// TIA Portal V15.1 export
// export: Created 2024-05-17T05:38:43.2423617Z, ExportSetting WithDefaults, DisplayName Totally Integrated Automation Portal, DisplayVersion V15.1 Update 5, DisplayName TIA Portal Openness, DisplayVersion V15.1 Update 5, DisplayName SINAMICS Startdrive Advanced, DisplayVersion V15.1, DisplayName G130, G150, S120, S150, SINAMICS MV, S210, DisplayVersion V15.1, DisplayName G110M, G120, G120C, G120D, G120P, DisplayVersion V15.1, DisplayName STEP 7 Professional, DisplayVersion V15.1 Update 5, DisplayName STEP 7 Safety, DisplayVersion V15.1, DisplayName WinCC Professional, DisplayVersion V15.1 Update 5, DisplayName SIMATIC Visualization Architect, DisplayVersion V15.1
FUNCTION "LGBShuttle5Pos2S-MoviFitFCPN-Config" : Void   // FC6696, FBD
TITLE = LMoveEPos-Config / LGBShuttle5Pos2S-MoviFitFCPN-Config
{ S7_Optimized_Access := 'FALSE' }
AUTHOR : VCC
FAMILY : Config
VERSION : 0.0.0.0
// =============================================================================
// Configuration MoveUnitEpos
// =============================================================================
// ============================================================================
// Configuration MoveUnitEpos
// ============================================================================
// stored: AutoNumber false, IsIECCheckEnabled false, SetENOAutomatically False, UDAEnableTagReadback false
   VAR_INPUT
      C_ForceManual : Bool;   // Force Manual Enabled
      C_AlarmResetUsed : Bool;   // Set position / If true, the Alarms will be stored untill reseted
      C_EnableMemBegin : Bool;   // Reset position / Enable memory Begin (Command Request is memorised until pos reached)
      C_EnIntlkAlm : Bool;   // Active / Enable interlock Alarm
      C_KeepPosition : Bool;   // Invisible / If true, the last position shall be kept ON and checked
      C_EnAlmOvertime : Bool;   // Object out of use / Enable Alarm
      C_InitDirection : Bool;   // Initial direction
      C_EnablePos1 : Bool;   // Position 1 used / Pos 1 used
      C_EnablePos2 : Bool;   // Position 2 used / Pos 2 used
      C_EnablePos3 : Bool;   // Position 3 used / Pos 3 used
      C_EnablePos4 : Bool;   // Position 4 used / Pos 4 used
      C_EnablePos5 : Bool;   // Position 5 used / Pos 4 used
      C_EnablePosMaint : Bool;   // Position Maintenance used / Pos 4 used
      C_SetHigherEncValue : Bool;   // Set direction to get HIGHER Encoder value
      C_OverTravelSetUsed : Bool;   // Overtravel set used
      C_OverTravelResUsed : Bool;   // Overtravel reset used
      C_MotorProtectionNc : Bool;   // Motor Protection NC contact
      C_MotorProtectionUsed : Bool;   // Motor Protection used
      C_MotionStopUsed : Bool;   // Motion Stop used
      C_HartingPlug400VNc : Bool;   // Motor Protection NC contact / Harting plug 400V NC contact
      C_HartingPlug400VUsed : Bool;   // Motor Protection used / Harting plug 400V used
      C_HartingPlug24VNc : Bool;   // Motor Protection NC contact / Harting plug 24V NC contact
      C_HartingPlug24VUsed : Bool;   // Motor Protection used / Harting plug 24V used
      C_EnableAlarmHW : Bool;   // Enable Alarm hardware (e.g. safetyswitch, motorprotector, detections)
      C_ReleaseBrakeUsed : Bool;   // Release brake used
      C_WhichPosIsHomePos : DInt;   // Which position is home position
      C_Pos1 : DInt;   // Position Stop 1
      C_Pos2 : DInt;   // Position Stop 2
      C_Pos3 : DInt;   // Position Stop 3
      C_Pos4 : DInt;   // Position Stop 4
      C_Pos5 : DInt;   // Position Stop 5 / Position Stop 4
      C_PosMaint : DInt;   // Maintenance Position
      C_Diff_HH_LL : DInt;   // Difference HH / LL
      C_Diff_H_L : DInt;   // Difference H / L
      C_RunTimeMaxSetWarn : DInt;   // Maximum Time (x1ms) that the function may run (create Overtime)
      C_RunTimeMaxSetAlarm : DInt;   // Maximum Time (x1ms) that the function may run (create Overtime)
      C_RunTimeMaxResWarn : DInt;   // Maximum Time (x1ms) that the function may run (create Overtime)
      C_RunTimeMaxResAlarm : DInt;   // Maximum Time (x1ms) that the function may run (create Overtime)
      C_TimeAlmFilt : DInt;   // Timer before any actuator Alarm will be active (welding..)
      C_Ramp : Time;   // Reference value for speed, stored in P2000 ot the SINAMICS / Configuration
      C_ReferenceDriveCurrent : Real;   // Drive reference current / Reference current of the drive
      C_ReferenceMotorCurrent : Real;   // Motor reference current / Reference current of the motor
      C_ReferenceMotorRPM : Real;   // Reference RPM of the motor
      C_RatioGearbox : Real;   // Acceleration in m/s²
      C_Diameter : Real;   // Diameter in mm
      C_Acceleration : Real;   // Ratio Gearbox <-> Motor
      C_HWSubInput : HW_SUBMODULE;   // I/O
      C_HWSubOutput : HW_SUBMODULE;   // I/O
      C_HWSubInputStatus : HW_SUBMODULE;   // I/O
   END_VAR
   VAR_IN_OUT
      IO_Config : "Shuttle5Pos2S-MoviFitFCPNConfig";   // Config
   END_VAR
BEGIN

REGION Network 1: **** 1 - Inputs **** Configuration / **** 1 - Inputs **** Move Bit Config
   // Configuration
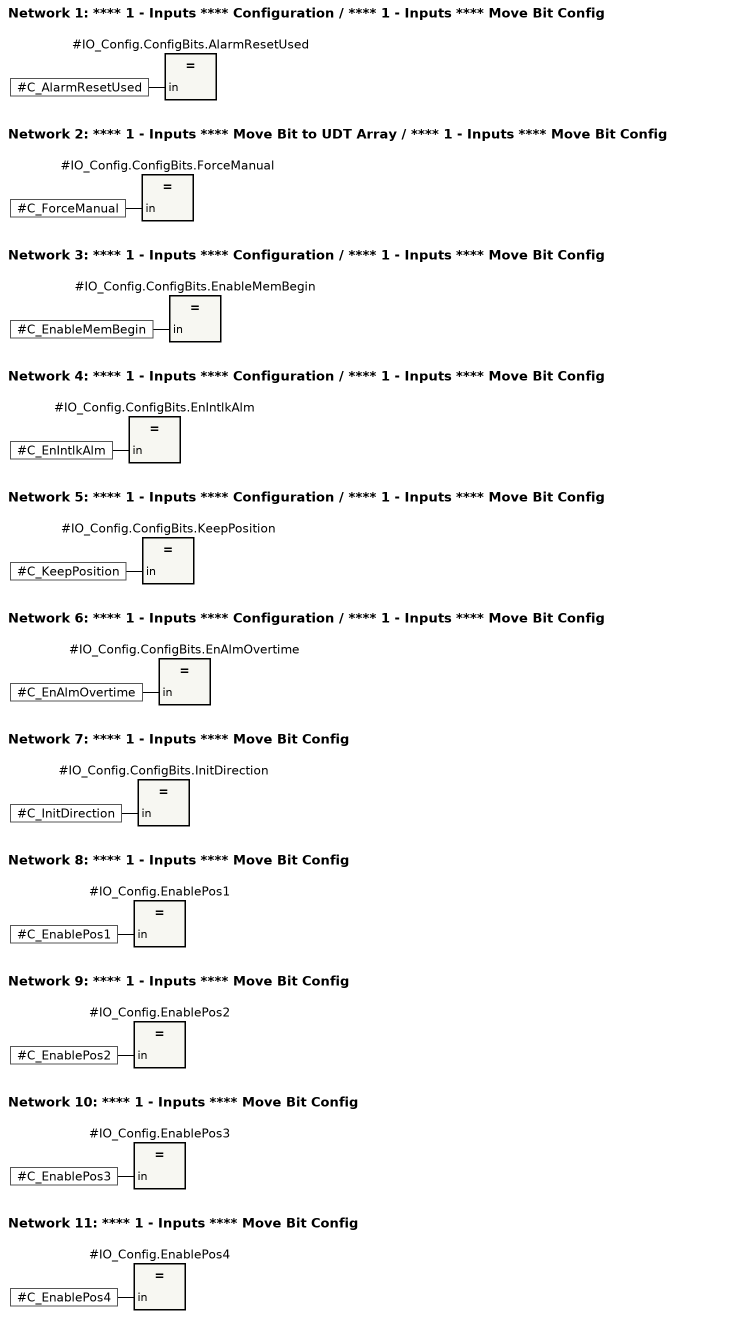
   #IO_Config.ConfigBits.AlarmResetUsed := #C_AlarmResetUsed;
END_REGION

REGION Network 2: **** 1 - Inputs **** Move Bit to UDT Array / **** 1 - Inputs **** Move Bit Config
   // Move Bit  to UDT Array
   #IO_Config.ConfigBits.ForceManual := #C_ForceManual;
END_REGION

REGION Network 3: **** 1 - Inputs **** Configuration / **** 1 - Inputs **** Move Bit Config
   // Configuration
   #IO_Config.ConfigBits.EnableMemBegin := #C_EnableMemBegin;
END_REGION

REGION Network 4: **** 1 - Inputs **** Configuration / **** 1 - Inputs **** Move Bit Config
   // Configuration
   #IO_Config.ConfigBits.EnIntlkAlm := #C_EnIntlkAlm;
END_REGION

REGION Network 5: **** 1 - Inputs **** Configuration / **** 1 - Inputs **** Move Bit Config
   // Configuration
   #IO_Config.ConfigBits.KeepPosition := #C_KeepPosition;
END_REGION

REGION Network 6: **** 1 - Inputs **** Configuration / **** 1 - Inputs **** Move Bit Config
   // Configuration
   #IO_Config.ConfigBits.EnAlmOvertime := #C_EnAlmOvertime;
END_REGION

REGION Network 7: **** 1 - Inputs **** Move Bit Config
   // Move Bit Config
   #IO_Config.ConfigBits.InitDirection := #C_InitDirection;
END_REGION

REGION Network 8: **** 1 - Inputs **** Move Bit Config
   // Move Bit Config
   #IO_Config.EnablePos1 := #C_EnablePos1;
END_REGION

REGION Network 9: **** 1 - Inputs **** Move Bit Config
   // Move Bit Config
   #IO_Config.EnablePos2 := #C_EnablePos2;
END_REGION

REGION Network 10: **** 1 - Inputs **** Move Bit Config
   // Move Bit Config
   #IO_Config.EnablePos3 := #C_EnablePos3;
END_REGION

REGION Network 11: **** 1 - Inputs **** Move Bit Config
   // Move Bit Config
   #IO_Config.EnablePos4 := #C_EnablePos4;
END_REGION

REGION Network 12: **** 1 - Inputs **** Move Bit Config
   // Move Bit Config
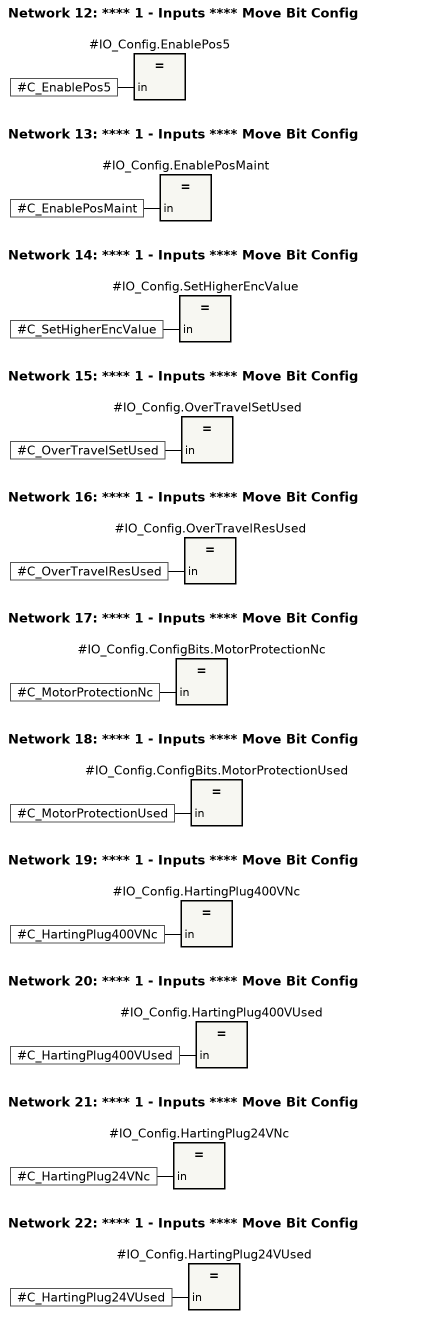
   #IO_Config.EnablePos5 := #C_EnablePos5;
END_REGION

REGION Network 13: **** 1 - Inputs **** Move Bit Config
   // Move Bit Config
   #IO_Config.EnablePosMaint := #C_EnablePosMaint;
END_REGION

REGION Network 14: **** 1 - Inputs **** Move Bit Config
   // Move Bit Config
   #IO_Config.SetHigherEncValue := #C_SetHigherEncValue;
END_REGION

REGION Network 15: **** 1 - Inputs **** Move Bit Config
   #IO_Config.OverTravelSetUsed := #C_OverTravelSetUsed;
END_REGION

REGION Network 16: **** 1 - Inputs **** Move Bit Config
   #IO_Config.OverTravelResUsed := #C_OverTravelResUsed;
END_REGION

REGION Network 17: **** 1 - Inputs **** Move Bit Config
   // Move Bit Config
   #IO_Config.ConfigBits.MotorProtectionNc := #C_MotorProtectionNc;
END_REGION

REGION Network 18: **** 1 - Inputs **** Move Bit Config
   // Move Bit Config
   #IO_Config.ConfigBits.MotorProtectionUsed := #C_MotorProtectionUsed;
END_REGION

REGION Network 19: **** 1 - Inputs **** Move Bit Config
   // Move Bit Config
   #IO_Config.HartingPlug400VNc := #C_HartingPlug400VNc;
END_REGION

REGION Network 20: **** 1 - Inputs **** Move Bit Config
   // Move Bit Config
   #IO_Config.HartingPlug400VUsed := #C_HartingPlug400VUsed;
END_REGION

REGION Network 21: **** 1 - Inputs **** Move Bit Config
   // Move Bit Config
   #IO_Config.HartingPlug24VNc := #C_HartingPlug24VNc;
END_REGION

REGION Network 22: **** 1 - Inputs **** Move Bit Config
   // Move Bit Config
   #IO_Config.HartingPlug24VUsed := #C_HartingPlug24VUsed;
END_REGION

REGION Network 23: **** 1 - Inputs **** Move Bit Config
   // Move Bit Config
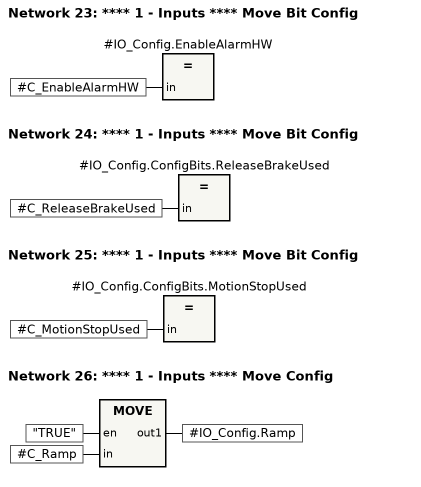
   #IO_Config.EnableAlarmHW := #C_EnableAlarmHW;
END_REGION

REGION Network 24: **** 1 - Inputs **** Move Bit Config
   // Move Bit Config
   #IO_Config.ConfigBits.ReleaseBrakeUsed := #C_ReleaseBrakeUsed;
END_REGION

REGION Network 25: **** 1 - Inputs **** Move Bit Config
   // Move Bit Config
   #IO_Config.ConfigBits.MotionStopUsed := #C_MotionStopUsed;
END_REGION

REGION Network 26: **** 1 - Inputs **** Move Config
   // Move Config
   IF "TRUE" THEN #IO_Config.Ramp := #C_Ramp; END_IF;
END_REGION

NETWORK
TITLE = **** 1 Inputs **** Move Config UDT
// Move Config
      L     #C_Diff_HH_LL;
      T     #IO_Config.Diff_HH_LL;
      L     #C_Diff_H_L;
      T     #IO_Config.Diff_H_L;
      L     #C_RunTimeMaxSetWarn;
      T     #IO_Config.RunTimeMaxSetWarn;
      L     #C_RunTimeMaxSetAlarm;
      T     #IO_Config.RunTimeMaxSetAlm;
      L     #C_RunTimeMaxResWarn;
      T     #IO_Config.RunTimeMaxResWarn;
      L     #C_RunTimeMaxResAlarm;
      T     #IO_Config.RunTimeMaxResAlm;
      L     #C_TimeAlmFilt;
      T     #IO_Config.TimeAlmFilt;
      L     #C_ReferenceMotorCurrent;
      T     #IO_Config.ReferenceMotorCurrent;
      L     #C_ReferenceMotorRPM;
      T     #IO_Config.ReferenceMotorRPM;
      L     #C_RatioGearbox;
      T     #IO_Config.RatioGearbox;
      L     #C_Diameter;
      T     #IO_Config.Diameter;
      L     #C_Acceleration;
      T     #IO_Config.Acceleration;
      L     #C_ReferenceDriveCurrent;
      T     #IO_Config.ReferenceDriveCurrent;
      L     #C_WhichPosIsHomePos;
      T     #IO_Config.WhichPosIsHomePos;
      L     #C_Pos1;
      T     #IO_Config.Pos1;
      L     #C_Pos2;
      T     #IO_Config.Pos2;
      L     #C_Pos3;
      T     #IO_Config.Pos3;
      L     #C_Pos4;
      T     #IO_Config.Pos4;
      L     #C_Pos5;
      T     #IO_Config.Pos5;
      L     #C_PosMaint;
      T     #IO_Config.PosMaint;
      L     #C_HWSubInput;
      T     #IO_Config.HWSubInput;
      L     #C_HWSubOutput;
      T     #IO_Config.HWSubOutput;
      L     #C_HWSubInputStatus;
      T     #IO_Config.HWSubInputStatus;
      NOP   0;
END_FUNCTION
